// TIA Portal V19 export
DATA_BLOCK "EDI DB"   // DB111
{ S7_Optimized_Access := 'FALSE' }
   VAR
      "EDI FEED PUMP 401ABC" : Bool;
      "EDI 501A" : Bool;
      "EDI 501B" : Bool;
      "AGLV-501 BUFF" : Int;
      "LEVEL HI RECIRC BUFF" : Int;
      "AGLV-501" : Bool;
      "AGLV-502" : Bool;
      "FLUSHING TIMER SET" : Int;
      "FLUSHING TIMER PV" : Int;
      "RECIRCULATION ON TIMER SET" : Int;
      "RECIRCULATION ON TIMER PV" : Int;
      "RECIRCULATION OFF TIMER SET" : Int;
      "RECIRCULATION OFF TIMER PV" : Int;
      "AGLV 501 FOR FLUSHING" : Bool;
      "AGLV 501 FOR RECIRCULATION" : Bool;
   END_VAR
BEGIN
END_DATA_BLOCK
